(* IEC 61131-3 sources: horner-cscape-mcp/artifacts/projects/TempTest/pous, 1 file *)

(* ---- TankLevelFailureTest.st ---- *)
PROGRAM TankLevelFailureTest
VAR
    TankLevel : REAL := 50.0;
    TargetLevel : REAL := 60.0;
END_VAR

TargetLevel := TankLevel + ;
END_PROGRAM
